(* IEC 61131-3 sources: repolevel_ST_code_completion/extract_code/轴控/FB101_功能块/F01_时钟脉冲, 3 files *)

(* ---- FB100ms时钟脉冲.st ---- *)
FUNCTION_BLOCK FB_100ms时钟脉冲
VAR_INPUT
	Input: BOOL;
END_VAR
VAR_OUTPUT
	Output: BOOL;
END_VAR
VAR
	TON1: TON;
	TON2: TON;
END_VAR

TON1(IN:= Input AND NOT TON2.Q, PT:= T#0.1S, Q=> , ET=> );
TON2(IN:= Input AND TON1.Q, PT:= T#0.1S, Q=> , ET=> );

IF TON1.Q THEN
	Output:=TRUE;
	ELSE
	Output:=FALSE;
END_IF

(* ---- FB500ms时钟脉冲.st ---- *)
FUNCTION_BLOCK FB_500ms时钟脉冲
VAR_INPUT
	Input: BOOL;
END_VAR
VAR_OUTPUT
	Output: BOOL;
END_VAR
VAR
	TON1: TON;
	TON2: TON;
END_VAR

TON1(IN:= Input AND NOT TON2.Q, PT:= T#0.5S, Q=> , ET=> );
TON2(IN:= Input AND TON1.Q, PT:= T#0.5S, Q=> , ET=> );

IF TON1.Q THEN
	Output:=TRUE;
	ELSE
	Output:=FALSE;
END_IF

(* ---- FB_时钟脉冲块.st ---- *)
FUNCTION_BLOCK FB_时钟脉冲块
(* Function block to simulate a turn signal *)
VAR_INPUT
	ENABLE:BOOL;		(* TRUE:run Blink, FALSE: OUT keeps its value*)
	TIMELOW:TIME;		(* Time for OUT=FALSE *)
	TIMEHIGH:TIME;		(* Time for OUT=TRUE *)
END_VAR
VAR_OUTPUT
	OUT:BOOL;			(* output variable, starting with FALSE *)
END_VAR
VAR
	CLOCK: TP;
END_VAR

CLOCK(IN:= ENABLE, PT:= , Q=> , ET=> );        (* call Timer *)

IF CLOCK.Q=FALSE AND ENABLE THEN            (* time passed or init *)
    CLOCK(IN:=FALSE);                       (* reset Timer *)
    CLOCK(IN:=TRUE);                        (* restart Timer *)
    IF OUT=FALSE THEN
        CLOCK.PT:=TIMEHIGH;
    ELSE
        CLOCK.PT:=TIMELOW;
    END_IF;
    OUT := NOT OUT;                         (* invert *)
END_IF
